(* IEC 61131-3 sources: ml2plc/benchmarks/st (part 15) *)

(* ---- MLP6.st ---- *)
FUNCTION_BLOCK MLP6_FB

    (* Model Inputs/Outputs *)
VAR_INPUT
    input_data : REAL;
END_VAR

VAR_OUTPUT
    output_data : ARRAY[0..2] OF REAL;
END_VAR

VAR CONSTANT
    weights_0 : ARRAY[0..31] OF REAL := [0.90454644, -0.400867403, 0.869943202, -0.168369889, -0.412142217, -0.709689677, 0.941532314, -0.0095654726, 0.967146814, -0.747319877, -0.0222444534, -0.66351074, -0.611298144, 1.09773886, -0.340438962, 1.20525312, 0.769771993, -0.182968155, -0.102920204, -0.384943873, -0.278610766, -0.314933598, 1.11625111, -0.168380052, -0.255054265, -0.366751343, -0.33793211, -0.02283746, 0.767741799, 0.474790365, 0.933169901, 0.962373257];
    bias_0 : ARRAY[0..31] OF REAL := [-0.170696706, 0, -0.161620259, 0, 0, 0.396536261, -0.158844277, 0, -0.152492061, 0.487909496, 0, 0.379839331, 0.448248148, -0.155945137, 0, -0.194220677, 0.0190808177, 0, 0, 0, 0, 0, 0.121851504, 0, 0, 0, 0.51204443, 0, -0.155369952, 0.399590701, -0.175982088, -0.155457303];

    weights_1 : ARRAY[0..767] OF REAL := [0.295231134, -0.129006118, 0.19198513, 1.21736336, -0.217146203, 0.906156719, -1.09466374, -0.706765652, 1.08418429, 0.564806283, 1.13035882, 0.892600179, -0.752894461, 1.10702014, 0.513110518, 0.785720646, -1.29299068, 0.0211936235, -1.44453084, -1.23774385, 1.08793128, -0.0487730801, -0.12848036, -1.00077665, 0.325005591, 0.290268898, 0.279054999, 0.285099328, -0.213655964, -0.16316177, 0.281590104, 0.239627063, 0.262345135, 0.0261963308, 0.0233350694, 0.294732571, 0.0434944928, 0.122584373, -0.150452822, -0.016712755, -0.261746407, -0.267375886, 0.240840673, -0.255916059, -0.249444306, 0.163675129, 0.0948724747, 0.162443012, 0.208322883, 0.238537252, -0.294643342, 1.23445666, -0.0170371439, 0.994598091, -0.975817561, -0.642093956, 1.19595969, 0.453583807, 1.12319052, 0.746419311, -0.853555024, 1.04991555, 0.597184777, 0.958240926, -1.17020535, 0.31369257, -1.47341204, -1.295645, 0.946281433, 0.27644223, -0.00174131989, -1.33688474, -0.176306188, -0.0927960575, 0.149620146, 0.286391616, -0.141670659, 0.0531999469, 0.153332919, 0.20505631, -0.167928115, 0.291448116, 0.150106311, -0.0987332314, 0.268482685, -0.307833642, 0.221213877, -0.321412444, 0.189507961, 0.191550195, 0.0819987059, -0.0778846443, 0.296701074, 0.225336492, 0.214712262, -0.0827709287, 0.285367191, -0.140551165, 0.00931853056, -0.138217196, 0.206591249, -0.0735297203, 0.221336126, 0.158516407, -0.0778366476, -0.271311015, 0.0633286238, -0.072303772, 0.108249843, -0.0929207653, -0.181190684, 0.0980706811, -0.0374506116, -0.320174545, 0.0739811957, -0.282686174, 0.186342359, 0.281644583, -0.259203553, 0.100598246, -0.0651429817, -0.206569076, -0.193545833, -0.482666612, -0.0821752772, -0.961810708, 1.172135, 0.69371134, -0.817266881, -0.412939996, -0.509167433, -0.866225541, 1.31189537, -0.633265257, -0.989419341, -0.846661031, 0.659452438, -0.225636706, 0.801334143, 0.350917637, -0.919107139, 0.225119472, -0.138609588, 0.721869826, -0.321482867, 0.123193502, 0.0898693502, 1.08808005, 0.295813471, 0.659393251, -0.476271152, -0.18717283, 1.23643327, 0.780925453, 0.986792803, 0.816414535, -0.891632259, 0.673117697, 0.646242201, 0.879625261, -0.865934372, -0.12343955, -1.18406153, -1.38234627, 0.901530623, 0.285107851, -0.256406724, -1.06379592, 0.107042551, 0.277778804, 0.193757594, 0.0590963066, -0.12765266, -0.133937359, -0.231395423, -0.289933264, 0.145242512, 0.23902446, 0.194817305, 0.0290448368, -0.0362384021, -0.17609328, 0.236915767, -0.0920998454, 0.252641916, 0.12115562, 0.000273287296, -0.269050717, -0.237204999, -0.219775066, 0.226729214, -0.231590211, -0.0661152154, -0.215537995, -0.235369325, 1.18310201, 0.173817322, 0.560130358, -0.859532833, -0.244359657, 1.11220109, 0.730377376, 0.526197612, 0.643959224, -0.431146711, 1.06084871, 0.894755185, 0.731103778, -0.696267724, 0.0121684372, -1.08033919, -1.12541819, 0.495167494, -0.101574555, 0.00402355194, -0.757044673, 0.136979058, 0.15508759, -0.02835216, -0.44361186, -0.275727361, -0.567569137, 0.871675193, 1.20000923, -0.853888154, -0.758741319, -0.443973094, -0.564651251, 1.32495701, -0.424292624, -0.405168772, -0.882857502, 0.919342339, -0.210148335, 0.787934899, 0.394117832, -0.723487794, -0.121570155, 0.274054289, 0.232991621, 0.184159577, -0.11905022, -0.173855618, 0.275910616, -0.213984191, 0.214573622, 0.247941315, -0.251989603, 0.207406044, 0.299859524, -0.0322960019, -0.235998034, -0.128714725, 0.137502581, -0.311281651, -0.0586145818, -0.236795753, 0.0351615846, -0.110103473, 0.0936356783, -0.203782856, 0.160411, -0.136357099, 0.217081785, -0.19382897, -0.0983214974, -0.172582373, -0.58115685, -0.227134705, -0.793690443, 0.987000167, 1.1088897, -0.533255935, -0.744200766, -0.41089806, -0.827442169, 0.908342123, -0.405829221, -0.716313243, -1.04521453, 0.604358673, -0.301062584, 0.378562003, 0.844146967, -0.835850179, 0.107833266, -0.223568857, 0.397432297, 0.188605264, -0.0674909353, 0.0566187575, 0.0197456405, 0.261059344, -0.524976611, 1.08699298, 1.06586397, -0.199344724, -0.802884936, -0.708495975, -0.716707826, 1.0185467, -0.364413172, -0.784771442, -0.431129128, 0.772798419, -0.185489476, 0.844132841, 0.761012673, -0.800541401, -0.0832273066, -0.2817581, 0.74396807, -0.264797121, -0.0910985023, -0.138044387, 0.990080476, 0.0802568346, 0.758434594, -0.552077353, -0.327732533, 0.887677908, 0.571260631, 0.937031686, 0.607444167, -0.378594458, 1.02893746, 0.491255462, 0.416121751, -1.0151366, -0.211483151, -0.746881902, -1.0333792, 0.443029851, -0.0171875358, -0.0381689072, -1.09573913, -0.043354094, 0.283042789, 0.206892252, 0.00916621089, -0.249695212, -0.295910805, 0.20259881, 0.162647396, 0.043733269, 0.20653832, -0.308564663, -0.280918926, 0.272660732, -0.172042117, 0.170747489, 0.23414731, 0.0630742013, 0.123369873, -0.207023829, 0.261101246, 0.213620901, 0.277589023, -0.0439403951, -0.205727562, 0.163603202, -0.113319919, -0.207964301, 0.628932774, -0.114935495, 0.705150783, -0.654717207, -0.237874627, 0.747101903, 0.727941096, 0.503591537, 0.72308296, -0.44854787, 0.965443373, 0.691107392, 0.5111745, -1.08201611, 0.21339798, -0.882919967, -1.20124686, 0.595513225, -0.252263993, 0.132210314, -1.06991637, -0.370881855, -0.0681702793, 0.169512168, 0.941228926, 0.070693031, 0.151429042, 0.256398469, 0.241526261, 0.751011312, 0.290890872, 0.30156377, 0.283818036, -0.0107974913, 0.482792228, 0.337298661, 0.281841606, -0.397284865, -0.208623588, -0.496294975, -0.470995426, 0.283237845, 0.0521007478, 0.144089073, -0.0686480999, -0.320380658, -0.277808845, 0.148536921, -0.0695285797, -0.277294815, -0.124862239, -0.0500250161, -0.222713381, -0.191136509, 0.246649325, 0.0220653415, 0.16214779, -0.061910063, 0.101160318, 0.157166272, -0.311789989, 0.000512182713, 0.0986146927, -0.171011031, 0.202872753, -0.215096593, -0.0623323619, -0.0904355496, 0.174473226, -0.301766038, 0.0454842746, -0.142736778, -0.020793587, -0.145345911, -0.178476349, 0.141361535, 0.0972788632, 0.110777199, 0.0764600039, 0.294599175, -2.27093697e-05, 0.173557222, 0.134258181, -0.311912924, -0.234820932, -0.187618434, -0.262826115, 0.192258656, 0.0524175763, 0.151788741, -0.03005898, 0.281539679, -0.157674417, -0.0799265057, -0.288467199, 0.0854136944, 0.153585076, 0.0907833874, -0.104148105, -0.0822955072, 0.210213959, 0.0297137201, -0.309015512, 0.0589160323, 0.156244159, -0.139795348, 0.276519597, 0.325013876, 0.0363880694, 0.127945542, 0.0618295372, -0.145081908, 0.192194581, 0.277251661, -0.144023046, -0.152517006, 0.231688559, -0.205610037, 0.22849232, 0.238232791, -0.29971382, 0.0167252421, -0.0997401178, -0.324124038, -0.127922207, 0.285681605, -0.10798724, -0.189939201, 0.294958234, -0.211431101, 0.211328328, -0.284518421, -0.18888253, -0.0722288787, -0.0350409448, -0.321308106, -0.0472274125, -0.0861286372, -0.316458166, -0.215742141, 0.0792055428, -0.0646136403, -0.274710715, -0.0250250399, -0.305008411, 0.229083359, 0.24799335, 0.0113067031, -0.249429077, -0.111249506, 0.237919688, -0.151925221, -0.318326861, -0.0953566432, 0.229551256, -0.163930863, 0.100224525, -0.167222232, -0.238116205, -0.202555746, -0.045360744, 0.0127826929, 0.280991137, -0.210080445, 0.0943366587, -0.0495974384, -0.0197191834, -0.149649471, 0.366648972, -0.281668693, 0.284846961, 0.403985202, 0.484802961, 0.784509182, 0.469572723, 0.473852932, 0.125889629, 0.312252492, 0.352212965, 0.477095902, -0.00642840099, -0.295710534, -0.206710175, -0.640399277, -0.231049523, 0.239183992, -0.311245203, -0.299947232, -0.0802108124, -0.0983978957, -0.173755497, -0.230084643, 0.316312313, -0.177855998, -0.298542112, 0.292203665, 0.00650158525, -0.297387481, -0.154374689, 0.162093848, 0.134812981, 0.246338308, 0.300070405, -0.310504198, -0.217782527, 0.0207454264, 0.0871799886, -0.264095902, 0.180105686, 0.285792828, 0.316828549, -0.150229871, 0.208020031, 0.136193275, -0.173812315, 0.0681842566, -0.221390352, 0.153097779, -0.194303483, 0.288291216, 0.12797904, 0.306318879, 0.212034047, -0.0300059021, 0.0768045485, -0.212660864, 0.171384782, 0.0894418657, -0.127920032, -0.21113494, -0.19953534, -0.211162567, 0.187122345, -0.174947098, -0.199379727, 0.0794975162, 0.270518363, 0.0516895354, 0.117571741, -0.0213138759, 0.146065593, -0.151934817, 0.324477196, 0.315924108, 0.0616651773, -0.300438493, 0.0912067592, -0.297835529, 0.13777557, 0.00982579589, -0.0171657801, -0.177937701, -0.210091144, 0.0937231779, -0.00284725428, -0.0512967706, -0.081265673, -0.277936608, 0.320349038, 0.0345208645, -0.0836495906, 0.218804076, -0.189922586, 0.00870514568, -0.0475570038, -0.215569362, -0.448498726, 0.7030285, 0.686182499, -0.145566911, -0.249483347, 0.0584986731, -0.39541024, 1.02209508, 0.23206374, -0.283743173, 0.0408624671, 0.087765269, 0.226524353, 0.406258434, 0.542207479, 0.000192098902, -0.154791355, -0.0193217993, 0.598222733, -0.155410215, -0.0176387131, -0.169864312, -0.207125589, -0.189757839, 0.0158335268, -0.170205817, 0.108427167, 0.163378179, 0.253302336, -0.147233725, -0.238223046, 0.0536537468, 0.00758227706, -0.275630891, 0.106042475, -0.240080804, -0.077775389, 0.144946277, -0.186762944, -0.104210451, 0.228787661, -0.0615751147, 0.211148441, -0.2518996, -0.019515574, 0.248782992, 1.05728996, -0.230006129, 0.742800951, -1.2359885, -0.62584269, 1.51240218, 0.719003975, 1.5774833, 0.910296917, -0.750651956, 1.05900729, 0.610199094, 1.06828773, -1.46972156, -0.31832701, -1.53218114, -1.44456565, 0.98592943, -0.268657327, -0.267539084, -1.16338086, -0.184921622, -0.0245098174, 0.181098208, 0.520282805, -0.0843829811, 0.0626276657, 0.461200267, 0.611355305, 0.621550381, -0.157471061, 0.200103998, -0.0395837352, 0.149573594, 0.173357353, -0.119783588, 0.0554200225, 0.0896117091, -0.160246953, 0.283200741, 0.299669445, -0.0905595943, -0.166233853, -0.0798888057, -0.229181871, 0.210135713, 0.0194011629, -0.0352008343, 0.728743076, 0.019356098, 0.761186361, -0.572355151, -0.597376704, 1.06806505, 0.662380099, 1.18272328, 0.938285351, -0.638570726, 0.836572111, 0.849231899, 0.980818689, -1.24159503, -0.29251948, -1.32303631, -1.02425313, 0.812224746, -0.230198115, 0.0245965719, -1.12541747, -0.0841034278, 0.118305951, 0.278894305, 1.19096649, 0.193239287, 0.558676004, -0.484399647, -0.12447723, 0.870661914, 0.808956504, 0.990534484, 0.965567052, -0.720074534, 0.667833567, 0.449974805, 0.92786181, -0.824072123, -0.092888996, -0.785955429, -0.710629821, 0.643768787, -0.179926112, -0.308975548, -0.589572847];
    bias_1 : ARRAY[0..23] OF REAL := [-0.041254133, 0, -0.00746029103, 0.0988344401, -0.0175108574, -0.163416371, 0.524258494, 0.51676178, 0.0377424657, -0.176874027, -0.0529647321, -0.118044838, 0.559266388, 0.0913945511, -0.158073679, -0.212183177, 0.239383668, 0, 0.26087296, 0.194069535, -0.150364339, 0, 0, 0.199199706];

    weights_2 : ARRAY[0..71] OF REAL := [-0.366981655, 0.407668054, -0.456144542, 0.0246128738, -0.193879545, 0.029107064, -0.161294922, 0.00702124368, -0.21840851, -1.41365981, 0.987270176, 0.742007971, -0.332335711, -0.0271744523, -0.441027492, -0.325576633, -1.88435066, 1.45009863, 0.876257122, 0.534476995, -1.14616477, 0.301283509, 0.361193687, -1.12447178, -1.20225334, 0.664745331, 0.887686074, -0.519799232, -1.71867156, 1.34296358, -1.97883332, 0.160939649, 0.910859942, -0.258056462, -1.82137454, 1.56507766, 0.472795397, 0.200812578, -1.2360208, -1.54919517, 0.81725806, 0.986340046, -0.0206529945, -1.71989512, 1.85158134, -0.0727280229, -1.53903365, 1.77559733, 1.76747835, -1.66802728, -0.428545892, -0.143300533, -0.339210212, 0.148096055, 1.281407, -2.03390622, -0.831091821, 1.72422087, -1.627334, -0.576684475, -0.803670168, -2.15200853, 1.69465089, 0.262259394, 0.242327183, 0.299449652, -0.337940395, -0.434468031, 0.11190328, 1.69577134, -2.20703983, -0.524324358];
    bias_2 : ARRAY[0..2] OF REAL := [0.173563749, 0.231935471, -0.377385825];

END_VAR

VAR
    (* Merged variables from all regions *)
    buffer_0 : ARRAY[0..23] OF REAL;
    buffer_1 : ARRAY[0..31] OF REAL;

    (* Temporary computation variables *)
    i : DINT;
    j : DINT;
    t : DINT;
    sum : REAL;
    (* Computation helpers *)
    max_val : REAL;
    exp_val : REAL;
    exp_sum : REAL;
    (* Spatial loop variables *)
    oc : DINT;
    oh : DINT;
    ow : DINT;
    ic : DINT;
    kh : DINT;
    kw : DINT;
    ih : DINT;
    iw : DINT;
END_VAR

(* Forward pass execution *)

(* Region: r0 [ACYCLIC] *)
(* Acyclic Region r0 *)
(* Layer 0: Fused Linear + RELU *)
FOR j := 0 TO 31 DO
    sum := 0.0;
    FOR i := 0 TO 0 DO
        sum := sum + input_data * weights_0[i * 32 + j];
    END_FOR;
buffer_1[j] := MAX(sum + bias_0[j], 0.0);
END_FOR;

(* Layer 1: Fused Linear + RELU *)
FOR j := 0 TO 23 DO
    sum := 0.0;
    FOR i := 0 TO 31 DO
        sum := sum + buffer_1[i] * weights_1[i * 24 + j];
    END_FOR;
buffer_0[j] := MAX(sum + bias_1[j], 0.0);
END_FOR;

(* Layer 2: Fused Linear + SOFTMAX *)
FOR j := 0 TO 2 DO
    sum := 0.0;
    FOR i := 0 TO 23 DO
        sum := sum + buffer_0[i] * weights_2[i * 3 + j];
    END_FOR;
output_data[j] := sum + bias_2[j];
END_FOR;

(* Softmax: find max *)
max_val := output_data[0];
FOR i := 1 TO 2 DO
    IF output_data[i] > max_val THEN
        max_val := output_data[i];
    END_IF;
END_FOR;

(* Softmax: compute exponentials and sum *)
exp_sum := 0.0;
FOR i := 0 TO 2 DO
    output_data[i] := EXP(output_data[i] - max_val);
    exp_sum := exp_sum + output_data[i];
END_FOR;

(* Softmax: normalize *)
FOR i := 0 TO 2 DO
    output_data[i] := output_data[i] / exp_sum;
END_FOR;

END_FUNCTION_BLOCK

(* ---- MLP6_straton.st ---- *)
FUNCTION_BLOCK MLP6_FB

    (* Model Inputs/Outputs *)
VAR_INPUT
    input_data : REAL;
END_VAR

VAR_OUTPUT
    output_data : ARRAY[0..2] OF REAL;
END_VAR

VAR
    CONSTANT weights_0 : ARRAY[0..31] OF REAL := [0.90454644, -0.400867403, 0.869943202, -0.168369889, -0.412142217, -0.709689677, 0.941532314, -0.0095654726, 0.967146814, -0.747319877, -0.0222444534, -0.66351074, -0.611298144, 1.09773886, -0.340438962, 1.20525312, 0.769771993, -0.182968155, -0.102920204, -0.384943873, -0.278610766, -0.314933598, 1.11625111, -0.168380052, -0.255054265, -0.366751343, -0.33793211, -0.02283746, 0.767741799, 0.474790365, 0.933169901, 0.962373257];
    CONSTANT bias_0 : ARRAY[0..31] OF REAL := [-0.170696706, 0, -0.161620259, 0, 0, 0.396536261, -0.158844277, 0, -0.152492061, 0.487909496, 0, 0.379839331, 0.448248148, -0.155945137, 0, -0.194220677, 0.0190808177, 0, 0, 0, 0, 0, 0.121851504, 0, 0, 0, 0.51204443, 0, -0.155369952, 0.399590701, -0.175982088, -0.155457303];
    CONSTANT weights_1 : ARRAY[0..767] OF REAL := [0.295231134, -0.129006118, 0.19198513, 1.21736336, -0.217146203, 0.906156719, -1.09466374, -0.706765652, 1.08418429, 0.564806283, 1.13035882, 0.892600179, -0.752894461, 1.10702014, 0.513110518, 0.785720646, -1.29299068, 0.0211936235, -1.44453084, -1.23774385, 1.08793128, -0.0487730801, -0.12848036, -1.00077665, 0.325005591, 0.290268898, 0.279054999, 0.285099328, -0.213655964, -0.16316177, 0.281590104, 0.239627063, 0.262345135, 0.0261963308, 0.0233350694, 0.294732571, 0.0434944928, 0.122584373, -0.150452822, -0.016712755, -0.261746407, -0.267375886, 0.240840673, -0.255916059, -0.249444306, 0.163675129, 0.0948724747, 0.162443012, 0.208322883, 0.238537252, -0.294643342, 1.23445666, -0.0170371439, 0.994598091, -0.975817561, -0.642093956, 1.19595969, 0.453583807, 1.12319052, 0.746419311, -0.853555024, 1.04991555, 0.597184777, 0.958240926, -1.17020535, 0.31369257, -1.47341204, -1.295645, 0.946281433, 0.27644223, -0.00174131989, -1.33688474, -0.176306188, -0.0927960575, 0.149620146, 0.286391616, -0.141670659, 0.0531999469, 0.153332919, 0.20505631, -0.167928115, 0.291448116, 0.150106311, -0.0987332314, 0.268482685, -0.307833642, 0.221213877, -0.321412444, 0.189507961, 0.191550195, 0.0819987059, -0.0778846443, 0.296701074, 0.225336492, 0.214712262, -0.0827709287, 0.285367191, -0.140551165, 0.00931853056, -0.138217196, 0.206591249, -0.0735297203, 0.221336126, 0.158516407, -0.0778366476, -0.271311015, 0.0633286238, -0.072303772, 0.108249843, -0.0929207653, -0.181190684, 0.0980706811, -0.0374506116, -0.320174545, 0.0739811957, -0.282686174, 0.186342359, 0.281644583, -0.259203553, 0.100598246, -0.0651429817, -0.206569076, -0.193545833, -0.482666612, -0.0821752772, -0.961810708, 1.172135, 0.69371134, -0.817266881, -0.412939996, -0.509167433, -0.866225541, 1.31189537, -0.633265257, -0.989419341, -0.846661031, 0.659452438, -0.225636706, 0.801334143, 0.350917637, -0.919107139, 0.225119472, -0.138609588, 0.721869826, -0.321482867, 0.123193502, 0.0898693502, 1.08808005, 0.295813471, 0.659393251, -0.476271152, -0.18717283, 1.23643327, 0.780925453, 0.986792803, 0.816414535, -0.891632259, 0.673117697, 0.646242201, 0.879625261, -0.865934372, -0.12343955, -1.18406153, -1.38234627, 0.901530623, 0.285107851, -0.256406724, -1.06379592, 0.107042551, 0.277778804, 0.193757594, 0.0590963066, -0.12765266, -0.133937359, -0.231395423, -0.289933264, 0.145242512, 0.23902446, 0.194817305, 0.0290448368, -0.0362384021, -0.17609328, 0.236915767, -0.0920998454, 0.252641916, 0.12115562, 0.000273287296, -0.269050717, -0.237204999, -0.219775066, 0.226729214, -0.231590211, -0.0661152154, -0.215537995, -0.235369325, 1.18310201, 0.173817322, 0.560130358, -0.859532833, -0.244359657, 1.11220109, 0.730377376, 0.526197612, 0.643959224, -0.431146711, 1.06084871, 0.894755185, 0.731103778, -0.696267724, 0.0121684372, -1.08033919, -1.12541819, 0.495167494, -0.101574555, 0.00402355194, -0.757044673, 0.136979058, 0.15508759, -0.02835216, -0.44361186, -0.275727361, -0.567569137, 0.871675193, 1.20000923, -0.853888154, -0.758741319, -0.443973094, -0.564651251, 1.32495701, -0.424292624, -0.405168772, -0.882857502, 0.919342339, -0.210148335, 0.787934899, 0.394117832, -0.723487794, -0.121570155, 0.274054289, 0.232991621, 0.184159577, -0.11905022, -0.173855618, 0.275910616, -0.213984191, 0.214573622, 0.247941315, -0.251989603, 0.207406044, 0.299859524, -0.0322960019, -0.235998034, -0.128714725, 0.137502581, -0.311281651, -0.0586145818, -0.236795753, 0.0351615846, -0.110103473, 0.0936356783, -0.203782856, 0.160411, -0.136357099, 0.217081785, -0.19382897, -0.0983214974, -0.172582373, -0.58115685, -0.227134705, -0.793690443, 0.987000167, 1.1088897, -0.533255935, -0.744200766, -0.41089806, -0.827442169, 0.908342123, -0.405829221, -0.716313243, -1.04521453, 0.604358673, -0.301062584, 0.378562003, 0.844146967, -0.835850179, 0.107833266, -0.223568857, 0.397432297, 0.188605264, -0.0674909353, 0.0566187575, 0.0197456405, 0.261059344, -0.524976611, 1.08699298, 1.06586397, -0.199344724, -0.802884936, -0.708495975, -0.716707826, 1.0185467, -0.364413172, -0.784771442, -0.431129128, 0.772798419, -0.185489476, 0.844132841, 0.761012673, -0.800541401, -0.0832273066, -0.2817581, 0.74396807, -0.264797121, -0.0910985023, -0.138044387, 0.990080476, 0.0802568346, 0.758434594, -0.552077353, -0.327732533, 0.887677908, 0.571260631, 0.937031686, 0.607444167, -0.378594458, 1.02893746, 0.491255462, 0.416121751, -1.0151366, -0.211483151, -0.746881902, -1.0333792, 0.443029851, -0.0171875358, -0.0381689072, -1.09573913, -0.043354094, 0.283042789, 0.206892252, 0.00916621089, -0.249695212, -0.295910805, 0.20259881, 0.162647396, 0.043733269, 0.20653832, -0.308564663, -0.280918926, 0.272660732, -0.172042117, 0.170747489, 0.23414731, 0.0630742013, 0.123369873, -0.207023829, 0.261101246, 0.213620901, 0.277589023, -0.0439403951, -0.205727562, 0.163603202, -0.113319919, -0.207964301, 0.628932774, -0.114935495, 0.705150783, -0.654717207, -0.237874627, 0.747101903, 0.727941096, 0.503591537, 0.72308296, -0.44854787, 0.965443373, 0.691107392, 0.5111745, -1.08201611, 0.21339798, -0.882919967, -1.20124686, 0.595513225, -0.252263993, 0.132210314, -1.06991637, -0.370881855, -0.0681702793, 0.169512168, 0.941228926, 0.070693031, 0.151429042, 0.256398469, 0.241526261, 0.751011312, 0.290890872, 0.30156377, 0.283818036, -0.0107974913, 0.482792228, 0.337298661, 0.281841606, -0.397284865, -0.208623588, -0.496294975, -0.470995426, 0.283237845, 0.0521007478, 0.144089073, -0.0686480999, -0.320380658, -0.277808845, 0.148536921, -0.0695285797, -0.277294815, -0.124862239, -0.0500250161, -0.222713381, -0.191136509, 0.246649325, 0.0220653415, 0.16214779, -0.061910063, 0.101160318, 0.157166272, -0.311789989, 0.000512182713, 0.0986146927, -0.171011031, 0.202872753, -0.215096593, -0.0623323619, -0.0904355496, 0.174473226, -0.301766038, 0.0454842746, -0.142736778, -0.020793587, -0.145345911, -0.178476349, 0.141361535, 0.0972788632, 0.110777199, 0.0764600039, 0.294599175, -2.27093697e-05, 0.173557222, 0.134258181, -0.311912924, -0.234820932, -0.187618434, -0.262826115, 0.192258656, 0.0524175763, 0.151788741, -0.03005898, 0.281539679, -0.157674417, -0.0799265057, -0.288467199, 0.0854136944, 0.153585076, 0.0907833874, -0.104148105, -0.0822955072, 0.210213959, 0.0297137201, -0.309015512, 0.0589160323, 0.156244159, -0.139795348, 0.276519597, 0.325013876, 0.0363880694, 0.127945542, 0.0618295372, -0.145081908, 0.192194581, 0.277251661, -0.144023046, -0.152517006, 0.231688559, -0.205610037, 0.22849232, 0.238232791, -0.29971382, 0.0167252421, -0.0997401178, -0.324124038, -0.127922207, 0.285681605, -0.10798724, -0.189939201, 0.294958234, -0.211431101, 0.211328328, -0.284518421, -0.18888253, -0.0722288787, -0.0350409448, -0.321308106, -0.0472274125, -0.0861286372, -0.316458166, -0.215742141, 0.0792055428, -0.0646136403, -0.274710715, -0.0250250399, -0.305008411, 0.229083359, 0.24799335, 0.0113067031, -0.249429077, -0.111249506, 0.237919688, -0.151925221, -0.318326861, -0.0953566432, 0.229551256, -0.163930863, 0.100224525, -0.167222232, -0.238116205, -0.202555746, -0.045360744, 0.0127826929, 0.280991137, -0.210080445, 0.0943366587, -0.0495974384, -0.0197191834, -0.149649471, 0.366648972, -0.281668693, 0.284846961, 0.403985202, 0.484802961, 0.784509182, 0.469572723, 0.473852932, 0.125889629, 0.312252492, 0.352212965, 0.477095902, -0.00642840099, -0.295710534, -0.206710175, -0.640399277, -0.231049523, 0.239183992, -0.311245203, -0.299947232, -0.0802108124, -0.0983978957, -0.173755497, -0.230084643, 0.316312313, -0.177855998, -0.298542112, 0.292203665, 0.00650158525, -0.297387481, -0.154374689, 0.162093848, 0.134812981, 0.246338308, 0.300070405, -0.310504198, -0.217782527, 0.0207454264, 0.0871799886, -0.264095902, 0.180105686, 0.285792828, 0.316828549, -0.150229871, 0.208020031, 0.136193275, -0.173812315, 0.0681842566, -0.221390352, 0.153097779, -0.194303483, 0.288291216, 0.12797904, 0.306318879, 0.212034047, -0.0300059021, 0.0768045485, -0.212660864, 0.171384782, 0.0894418657, -0.127920032, -0.21113494, -0.19953534, -0.211162567, 0.187122345, -0.174947098, -0.199379727, 0.0794975162, 0.270518363, 0.0516895354, 0.117571741, -0.0213138759, 0.146065593, -0.151934817, 0.324477196, 0.315924108, 0.0616651773, -0.300438493, 0.0912067592, -0.297835529, 0.13777557, 0.00982579589, -0.0171657801, -0.177937701, -0.210091144, 0.0937231779, -0.00284725428, -0.0512967706, -0.081265673, -0.277936608, 0.320349038, 0.0345208645, -0.0836495906, 0.218804076, -0.189922586, 0.00870514568, -0.0475570038, -0.215569362, -0.448498726, 0.7030285, 0.686182499, -0.145566911, -0.249483347, 0.0584986731, -0.39541024, 1.02209508, 0.23206374, -0.283743173, 0.0408624671, 0.087765269, 0.226524353, 0.406258434, 0.542207479, 0.000192098902, -0.154791355, -0.0193217993, 0.598222733, -0.155410215, -0.0176387131, -0.169864312, -0.207125589, -0.189757839, 0.0158335268, -0.170205817, 0.108427167, 0.163378179, 0.253302336, -0.147233725, -0.238223046, 0.0536537468, 0.00758227706, -0.275630891, 0.106042475, -0.240080804, -0.077775389, 0.144946277, -0.186762944, -0.104210451, 0.228787661, -0.0615751147, 0.211148441, -0.2518996, -0.019515574, 0.248782992, 1.05728996, -0.230006129, 0.742800951, -1.2359885, -0.62584269, 1.51240218, 0.719003975, 1.5774833, 0.910296917, -0.750651956, 1.05900729, 0.610199094, 1.06828773, -1.46972156, -0.31832701, -1.53218114, -1.44456565, 0.98592943, -0.268657327, -0.267539084, -1.16338086, -0.184921622, -0.0245098174, 0.181098208, 0.520282805, -0.0843829811, 0.0626276657, 0.461200267, 0.611355305, 0.621550381, -0.157471061, 0.200103998, -0.0395837352, 0.149573594, 0.173357353, -0.119783588, 0.0554200225, 0.0896117091, -0.160246953, 0.283200741, 0.299669445, -0.0905595943, -0.166233853, -0.0798888057, -0.229181871, 0.210135713, 0.0194011629, -0.0352008343, 0.728743076, 0.019356098, 0.761186361, -0.572355151, -0.597376704, 1.06806505, 0.662380099, 1.18272328, 0.938285351, -0.638570726, 0.836572111, 0.849231899, 0.980818689, -1.24159503, -0.29251948, -1.32303631, -1.02425313, 0.812224746, -0.230198115, 0.0245965719, -1.12541747, -0.0841034278, 0.118305951, 0.278894305, 1.19096649, 0.193239287, 0.558676004, -0.484399647, -0.12447723, 0.870661914, 0.808956504, 0.990534484, 0.965567052, -0.720074534, 0.667833567, 0.449974805, 0.92786181, -0.824072123, -0.092888996, -0.785955429, -0.710629821, 0.643768787, -0.179926112, -0.308975548, -0.589572847];
    CONSTANT bias_1 : ARRAY[0..23] OF REAL := [-0.041254133, 0, -0.00746029103, 0.0988344401, -0.0175108574, -0.163416371, 0.524258494, 0.51676178, 0.0377424657, -0.176874027, -0.0529647321, -0.118044838, 0.559266388, 0.0913945511, -0.158073679, -0.212183177, 0.239383668, 0, 0.26087296, 0.194069535, -0.150364339, 0, 0, 0.199199706];
    CONSTANT weights_2 : ARRAY[0..71] OF REAL := [-0.366981655, 0.407668054, -0.456144542, 0.0246128738, -0.193879545, 0.029107064, -0.161294922, 0.00702124368, -0.21840851, -1.41365981, 0.987270176, 0.742007971, -0.332335711, -0.0271744523, -0.441027492, -0.325576633, -1.88435066, 1.45009863, 0.876257122, 0.534476995, -1.14616477, 0.301283509, 0.361193687, -1.12447178, -1.20225334, 0.664745331, 0.887686074, -0.519799232, -1.71867156, 1.34296358, -1.97883332, 0.160939649, 0.910859942, -0.258056462, -1.82137454, 1.56507766, 0.472795397, 0.200812578, -1.2360208, -1.54919517, 0.81725806, 0.986340046, -0.0206529945, -1.71989512, 1.85158134, -0.0727280229, -1.53903365, 1.77559733, 1.76747835, -1.66802728, -0.428545892, -0.143300533, -0.339210212, 0.148096055, 1.281407, -2.03390622, -0.831091821, 1.72422087, -1.627334, -0.576684475, -0.803670168, -2.15200853, 1.69465089, 0.262259394, 0.242327183, 0.299449652, -0.337940395, -0.434468031, 0.11190328, 1.69577134, -2.20703983, -0.524324358];
    CONSTANT bias_2 : ARRAY[0..2] OF REAL := [0.173563749, 0.231935471, -0.377385825];
END_VAR

VAR
    (* Merged variables from all regions *)
    buffer_0 : ARRAY[0..23] OF REAL;
    buffer_1 : ARRAY[0..31] OF REAL;

    (* Temporary computation variables *)
    i : DINT;
    j : DINT;
    t : DINT;
    sum : REAL;
    (* Computation helpers *)
    max_val : REAL;
    exp_val : REAL;
    exp_sum : REAL;
    (* Spatial loop variables *)
    oc : DINT;
    oh : DINT;
    ow : DINT;
    ic : DINT;
    kh : DINT;
    kw : DINT;
    ih : DINT;
    iw : DINT;
END_VAR

(* Forward pass execution *)

(* Region: r0 [ACYCLIC] *)
(* Acyclic Region r0 *)
(* Layer 0: Fused Linear + RELU *)
FOR j := 0 TO 31 DO
    sum := 0.0;
    FOR i := 0 TO 0 DO
        sum := sum + input_data * weights_0[i * 32 + j];
    END_FOR;
buffer_1[j] := MAX(sum + bias_0[j], 0.0);
END_FOR;

(* Layer 1: Fused Linear + RELU *)
FOR j := 0 TO 23 DO
    sum := 0.0;
    FOR i := 0 TO 31 DO
        sum := sum + buffer_1[i] * weights_1[i * 24 + j];
    END_FOR;
buffer_0[j] := MAX(sum + bias_1[j], 0.0);
END_FOR;

(* Layer 2: Fused Linear + SOFTMAX *)
FOR j := 0 TO 2 DO
    sum := 0.0;
    FOR i := 0 TO 23 DO
        sum := sum + buffer_0[i] * weights_2[i * 3 + j];
    END_FOR;
output_data[j] := sum + bias_2[j];
END_FOR;

(* Softmax: find max *)
max_val := output_data[0];
FOR i := 1 TO 2 DO
    IF output_data[i] > max_val THEN
        max_val := output_data[i];
    END_IF;
END_FOR;

(* Softmax: compute exponentials and sum *)
exp_sum := 0.0;
FOR i := 0 TO 2 DO
    output_data[i] := EXP(output_data[i] - max_val);
    exp_sum := exp_sum + output_data[i];
END_FOR;

(* Softmax: normalize *)
FOR i := 0 TO 2 DO
    output_data[i] := output_data[i] / exp_sum;
END_FOR;

END_FUNCTION_BLOCK

(* ---- MLP7.st ---- *)
FUNCTION_BLOCK MLP7_FB

    (* Model Inputs/Outputs *)
VAR_INPUT
    input_data : REAL;
END_VAR

VAR_OUTPUT
    output_data : ARRAY[0..2] OF REAL;
END_VAR

VAR CONSTANT
    weights_0 : ARRAY[0..23] OF REAL := [-0.0746802986, 0.607636034, 0.455998242, 0.258762628, -0.13258031, 0.252115637, -0.10976994, 0.548266053, -0.441276819, -0.438432246, 0.647188544, 0.493570745, -0.43271625, -0.082831949, 0.649822593, 0.439375341, -0.287549376, -0.311959922, 0.274157524, 0.315673918, 0.643515408, -0.171732515, 0.496268243, -0.371054083];
    bias_0 : ARRAY[0..23] OF REAL := [0, -0.12941812, -0.105221123, -0.0604603514, 0, 0.207637087, 0, 0.0315683261, 0, 0, -0.117396198, -0.0605233088, 0, 0, 0.0510026328, -0.0530445352, 0, 0, -0.0639983788, 0.203389689, -0.111548714, 0, -0.0640599579, 0];

    weights_1 : ARRAY[0..575] OF REAL := [-0.268907338, 0.00217190385, 0.137464732, -0.0683488548, -0.0738091469, 0.0699335039, -0.0417425632, 0.19087711, 0.0489356816, 0.344365627, 0.157603174, 0.211316198, -0.259004354, -0.257717103, 0.277782112, 0.273165613, 0.265473157, -0.205595359, 0.217125148, 0.343775719, 0.000431239605, -0.204861492, -0.16889219, -0.295836747, -0.612856627, -0.141135335, 0.4472965, -0.0880493671, -0.0630476475, -0.510043383, 0.529629707, 0.314925313, -0.324320614, -0.509671628, 0.322658747, 0.241676986, 0.696524978, 0.524104714, -0.213002667, 0.243135035, -0.297149271, -0.177744299, -0.219710499, 0.546750069, 0.511470258, 0.148470536, 0.587771058, 0.699641109, -0.699686229, -0.0136144357, 0.265989453, 0.187910274, 0.342317551, -0.476634353, 0.119458191, -0.123250976, 0.135319307, -0.525157869, -0.262663037, 0.386619776, 0.15526025, 0.15252319, 0.0138672292, 0.709074318, -0.214552373, 0.198164448, -0.329590023, 0.262734801, 0.253178746, 0.00747139985, 0.705926538, 0.132839769, -0.604175448, 0.0361758061, 0.386252105, 0.259136945, 0.121620715, -0.502793372, 0.120056905, 0.172273502, 0.197177142, -0.220736131, 0.312253743, 0.319560826, 0.478767067, 0.399403363, 0.299865872, 0.712916255, 0.00703683496, -0.358783484, -0.118123114, 0.141307041, 0.27085793, -0.305572391, 0.74335593, 0.179063112, -0.300123811, 0.294067651, 0.277188748, -0.273958385, -0.176085144, -0.0395295322, 0.172060519, -0.157897264, -0.331464142, -0.019657284, 0.114273429, 0.14408347, 0.0497518182, -0.119545832, -0.169999823, -0.30714044, -0.0324544311, 0.29038915, 0.094248265, 0.210150927, 0.158477634, -0.136283606, -0.0214261115, 0.0398223698, 0.216942891, -0.0235428363, 0.118681543, 0.083537966, -0.249544412, 0.332191288, 0.358593881, -0.315374881, 0.236496851, 0.186359823, -0.021189332, 0.485366553, -0.218409613, -0.00703188404, -0.112409517, -0.153913006, 0.210461989, 0.118319869, 0.173140079, 0.35994482, 0.224077418, 0.377764165, 0.135184735, 0.0969982445, 0.0219076872, -0.319111407, 0.0442451835, 0.314922959, 0.342028826, 0.154806107, -0.251459479, 0.231669575, 0.166534096, -0.14645718, -0.199890018, 0.29779157, 0.181536824, 0.22370407, 0.147348255, -0.241052836, 0.276352018, 0.0678429306, -0.271346122, -0.32665199, -0.179163054, 0.057913214, -0.216329142, -0.161545247, 0.236314058, 0.198999107, 0.204323336, 0.109188184, 0.185613602, -0.00481222663, -0.108478963, -0.184006527, -0.16169177, -0.126572222, -0.182018921, 0.401931792, 0.0411342047, 0.274655849, -0.312093377, 0.0779248402, -0.244552612, -0.0933865234, -0.143112406, 0.316888869, -0.0897234753, 0.444688708, 0.0414355583, 0.468671679, 0.224688619, -0.106085896, 0.12706238, 0.0274204016, -0.269548059, 0.0074904263, -0.25059554, -0.250605166, 0.317630261, 0.123651862, -0.246514887, 0.168738812, 0.28361252, 0.119744748, 0.141637355, 0.193590432, 0.245099097, -0.271869928, 0.305476636, 0.214189082, 0.0639041364, -0.251134604, -0.280500591, -0.182719231, 0.0889582634, 0.106302857, 0.308100551, -0.123537555, 0.155842453, 0.0435905457, 0.282452852, 0.0464273691, -0.329868048, 0.189582318, 0.0826188624, 0.268325478, -0.282127619, 0.325057715, 0.0578409731, -0.106060609, 0.122288734, 0.281878263, 0.0715391338, 0.0967436135, 0.312681288, 0.346843749, 0.286530644, 0.323031157, -0.62107712, 0.31202659, 0.439596415, -0.344784915, -0.217742249, -0.058255773, 0.255871952, 0.122528382, 0.234015152, 0.190027699, 0.0680105984, 0.477807403, 0.580108285, 0.111387841, 0.32501927, 0.465298355, 0.0707894638, 0.211896211, 0.313886732, 0.0590125956, 0.536113501, -0.110482946, 0.383503079, 0.321528226, -0.391103178, -0.0757583752, 0.477379769, -0.0182638038, -0.226764709, -0.114267945, 0.544339299, 0.341566026, 0.204276666, -0.276710838, -0.0310451984, 0.337987483, 0.101955645, 0.466226697, 0.00610649586, 0.0666570589, 0.251989096, -0.0348885134, -0.029322058, 0.0374343842, 0.548539996, 0.448163837, -0.0839401558, 0.467522532, -0.0633949339, 0.207616359, 0.0878649652, 0.00687465072, 0.266888529, 0.191955179, -0.319217205, 0.33818987, 0.0626723766, -0.093282342, 0.290955514, -0.015552938, -0.147785395, -0.222969472, 0.000421226025, 0.087808311, -0.184572592, -0.030451268, 0.308537692, 0.324173838, -0.0962346494, -0.0917209089, 0.121005028, 0.0796872079, 0.212975711, -0.169214532, -0.0300399065, 0.26500538, 0.0404863358, 0.188591808, -0.195912629, 0.175725371, -0.119754195, -0.180573285, -0.260601789, 0.318698615, 0.0112495124, 0.332248241, -0.0760537386, -0.140548617, 0.0673505664, 0.277959973, -0.230266511, -0.304319382, -0.0186672509, -0.289335996, 0.174558014, -0.0480471551, 0.156338379, -0.338227391, 0.379409701, -0.329904109, -0.0335883498, -0.0243462808, 0.106674857, -0.207976103, -0.31758371, -0.205548838, -0.286922336, 0.453636765, 0.344143778, -0.139424697, 0.150888771, 0.368412137, -0.0207992848, 0.433938384, -0.227954015, 0.451291412, 0.0406967625, 0.444359481, 0.183337077, 0.00309645641, 0.182288632, 0.142382234, -0.138220325, -0.0159723535, -0.266371191, -0.157991484, 0.509245634, -0.3441737, -0.300116122, -0.289941072, -0.25277108, 0.275200456, 0.381681621, 0.368882239, 0.191403657, 0.299521059, 0.0331215486, 0.0199813955, 0.0838560462, -0.0338563249, 0.552538455, -0.0257612541, 0.162927568, 0.157294571, -0.0424414575, 0.0741851032, 0.00993341208, 0.14510569, -0.19807291, -0.216219321, -0.326386631, -0.0369665921, -0.350637496, 0.327333599, 0.187157542, -0.191772714, -0.272784531, 0.178999513, 0.170922011, 0.344064087, 0.273409277, -0.195383936, 0.0219087601, -0.320345551, -0.223053589, -0.167534485, -0.353014231, -0.0325659513, 0.133774012, 0.300787896, -0.154813468, -0.109787136, 0.0450620651, -0.120923176, -0.126991063, -0.150874168, 0.330428869, -0.0456075966, 0.0592706203, 0.153212577, -0.167818964, -0.31344831, -0.313499629, 0.0622265339, -0.132025421, -0.0950550437, -0.172515988, -0.309438348, -0.241304442, 0.0670445859, 0.340844244, -0.00674307346, -0.0571297407, 0.195944682, 0.291546017, -0.089925617, -0.17480801, -0.509736598, 0.418891937, 0.187606826, -0.153403401, -0.149088994, 0.208767861, -0.081951119, 0.658967853, 0.617743134, -0.0702296197, 0.572496474, 0.191262931, 0.193394378, -0.252258331, 0.573703945, 0.182828963, -0.104402117, 0.189143315, 0.72547698, 0.252746373, -0.127337083, 0.359964609, 0.252452195, 0.0182416737, 0.158887416, 0.348938584, -0.0390769318, 0.164680511, 0.340248942, -0.29226917, -0.0991819948, 0.165644377, -0.00725150527, -0.105002299, -0.112420052, -0.139867827, 0.569023848, -0.310940892, 0.0389346555, 0.177371755, 0.124769427, 0.120482311, -0.127293751, 0.0575004928, -0.217616215, 0.0183300879, 0.123401649, 0.098418802, -0.383335978, 0.410907269, -0.0536490418, -0.247322127, -0.27997908, 0.27313289, 0.325315207, 0.4671942, 0.590981603, -0.332647026, 0.412228435, -0.349655986, -0.245886207, -0.194440514, 0.346960187, 0.216047853, 0.107523225, 0.0693727285, 0.547360241, -0.303221017, -0.0726420283, -0.102691054, 0.24672243, 0.184002489, -0.106598735, -0.143918335, 0.0378342271, 0.105892092, -0.0521823466, -0.241860956, 0.0522222221, 0.290780276, 0.329312891, -0.0297322273, 0.299719065, -0.0803425908, -0.127563834, -0.258438736, 0.128532708, 0.0761955082, 0.202705115, -0.275218487, 0.284864634, -0.285524696, 0.23296684, 0.558344007, -0.370309085, 0.0632788539, -0.199879572, 0.378469765, 0.168243155, -0.204663306, -0.111090496, -0.0149026215, 0.482993186, 0.230562359, -0.0151113905, -0.081802994, 0.302559614, 0.28712967, 0.350448579, 0.287046105, 0.0832951739, 0.450847089, 0.149081931, 0.352454573, 0.548047662, -0.231863469, 0.299252719, -0.0325100422, -0.237312376, 0.0971217752, -0.00699299574, 0.248950452, -0.0907193124, -0.16760385, 0.145382762, 0.0910830498, -0.00387185812, -0.277013451, 0.126328528, -0.23418954, -0.0778735578, -0.27938059, -0.349283576, 0.0730948448, 0.255102366, 0.0797807872, 0.0635040104, 0.0545716584, 0.144961387];
    bias_1 : ARRAY[0..23] OF REAL := [0.176716387, -0.00299654785, 0.0593073107, -0.0575258322, 0, 0.129074454, -0.103701882, -0.0082479585, -0.0571199395, 0.0882943869, 0, 0.208057463, -0.135922343, -0.0881750807, 0, -0.0836111233, -0.00893536955, 0.244989246, 0, -0.100842871, 0.0560074486, 0.252564728, -0.143066466, -0.12537545];

    weights_2 : ARRAY[0..575] OF REAL := [-0.245642945, -0.246756554, -0.328891218, -0.563465476, -0.555797517, 0.0490016043, -0.233312637, -0.150199234, 0.353149563, -0.227947727, 0.0115364343, 0.158489317, 0.142654747, -0.431395471, 0.344945014, 0.324086517, 0.612027287, -0.219665155, -0.0898557678, 0.145038947, 0.593772233, -0.217062712, -0.195034459, -0.363241315, 0.119104199, 0.22720471, -0.0466149151, -0.0383172072, -0.331802279, 0.343306452, -0.171254784, 0.156157047, 0.276797444, 0.220166475, -0.158973664, 0.32375142, 0.0450913534, -0.326723188, -0.201807857, 0.308251947, 0.226838693, 0.0587440133, 0.245269522, 0.266734153, 0.1890876, 0.0765732601, -0.0288925171, 0.223519564, 0.280389965, 0.0145830512, 0.00144499971, 0.139997378, 0.113765299, -0.191146329, 0.307509392, 0.179293185, 0.374915421, 0.30121091, 0.495148122, 0.0815368593, 0.434390634, -0.14555715, 0.433478117, -0.190034807, -0.0800786242, -0.200110286, 0.509086668, 0.318211406, 0.302050829, 0.0287599247, 0.141590983, 0.31887728, -0.226454079, 0.348596007, -0.016703397, 0.173407003, -0.270399421, 0.0868661702, -0.156372473, -0.12866497, 0.372414291, 0.347522587, 0.182157025, 0.241545171, -0.323187351, -0.271822125, -0.0328329206, -0.257270426, 0.004878846, -0.164576188, 0.32456243, 0.324977875, -0.0877593905, 0.244203418, 0.17296055, -0.27077353, -0.148512006, 0.0627348125, -0.235144854, 0.224023789, 0.258846492, 0.190566212, -0.136538416, 0.244612128, -0.260796845, -0.264053375, 0.20704934, 0.112125605, 0.108366191, 0.0839831531, -0.248119086, 0.210814208, -0.126879886, -0.19144927, -0.0575715005, -0.315923661, 0.152904361, -0.107165188, 0.098418355, -0.281930566, -0.0221283156, -0.242865384, 0.147830218, -0.0177736022, -0.0663293079, -0.191042975, -0.139932171, -0.0271336436, 0.306826115, 0.108970776, -0.47794044, 0.289082974, 0.848751605, -0.043951571, 0.271782011, 0.565594852, 0.176920876, 0.293638378, -0.185994714, -0.183791861, 0.492481083, -0.160842761, -0.195042297, -0.15548411, 0.224055469, 0.200847, -0.0932983235, 0.251617342, 0.455671281, 0.261954457, -0.0860045254, -0.0112277567, 0.242849126, -0.0363826528, 0.0945869535, -0.158523649, 0.232608065, 0.18994756, 0.048118569, 0.226275221, -0.00935058389, -0.233899072, -0.0633342341, 0.261702985, 0.00170290633, 0.43676585, -0.244740173, 0.53414011, 0.204737216, -0.0611152947, -0.105342865, -0.0732150078, 0.120023869, 0.261113197, 0.138036996, 0.333630413, 0.250143796, -0.0457339585, 0.214532509, -0.307090104, -0.333172113, 0.0266219284, -0.334947944, 0.0495177507, -0.121425427, 0.226054937, 0.281170636, 0.107468642, 0.277073115, -0.225816518, -0.219915509, -0.15749234, 0.184502214, -0.273863554, 0.233854562, -0.0685526431, -0.291586995, 0.0733211935, -0.303754866, 0.266844183, 0.311533213, 0.295593113, 0.183031395, 0.138876736, -0.298650354, 0.187308699, 0.158070579, -0.038877558, -0.0276067965, -0.141152993, 0.110567927, -0.232558206, -0.186817855, 0.0793989003, -0.158586457, 0.22946766, -0.501852512, -0.299868256, 0.256566316, -0.582294166, -0.448347151, -0.210635707, 0.322008342, -0.258173883, 0.379928738, 0.275341272, 0.199535474, -0.322017342, 0.800383627, -0.195558012, 0.220077574, 0.16850391, 0.0875466466, -0.137633145, -0.405929536, 0.0637919232, 0.397787511, -0.118515283, -0.0634722114, -0.508549154, -0.318264753, -0.0369980335, 0.339129716, -0.185298115, 0.318987221, -0.257021844, 0.326296836, -0.125292212, 0.215666503, 0.00417363644, -0.105437919, 0.0311455131, -0.263626844, 0.0762697756, -0.0561151505, 0.2861332, -0.207532167, 0.3018938, 0.0366989374, 0.210771888, -0.133724362, 0.0648821294, 0.0861230493, -0.151588723, 0.165128812, -0.318110764, 0.0824543834, 0.410491556, -0.16636388, -0.265668929, -0.217291281, -0.280920208, 0.376858443, -0.303223848, 0.448855996, -0.170281783, 0.354806125, 0.0322148241, 0.419946581, -0.099502638, 0.0150394971, -0.224528477, 0.499678612, 0.0742175803, 0.185917586, 0.272458673, -0.24160108, -0.0894065127, 0.669480681, -0.0906793773, 0.0840942785, 0.293848902, 0.649855793, -0.118749589, -0.319913119, 0.00412905216, -0.229158893, 0.131725997, 0.490128577, 0.209284037, -0.309097946, 0.35574317, 0.25872305, -0.335510433, -0.425682485, -0.228162214, 0.511070549, 0.0847743154, -0.507714033, 0.37029779, -0.130451664, 0.461581945, 0.503590107, -0.0959527791, -0.10381075, 0.129085854, 0.118843004, -0.0449370444, 0.265093714, 0.138016343, -0.413666576, 0.185948581, 0.289212912, -0.0518284738, -0.188458264, 0.396242261, -0.00943513215, -0.649417937, -0.62592417, 0.00135046244, 0.452810377, 0.501355469, -0.709819973, 0.628315389, 0.343882769, 0.65114969, -0.0102708638, -0.16960068, 0.320089728, 0.325349718, -0.327407748, 0.243835896, -0.0235780478, 0.210580379, 0.239429086, -0.0277884305, 0.245251507, -0.0667792261, 0.0719113648, 0.226514786, -0.228350446, -0.214209169, 0.0621877611, 0.307303458, -0.116270259, -0.338030607, -0.0395987332, -0.278134644, -0.0744503736, 0.297008485, 0.393869758, 0.33913973, 0.12972188, 0.293395817, 0.713052988, 0.037013948, -0.172523066, 0.0210779905, -0.549971342, 0.0169248395, 0.0676543564, -0.078420192, -0.274449199, 0.307433218, 0.00872946065, -0.376850694, -0.411587656, 0.106564432, 0.32417807, 0.567158878, -0.647322595, 0.517194271, 0.351190478, 0.386148691, 0.324564457, -0.349219918, 0.0146075785, 0.341831416, 0.135289431, -0.112718031, -0.0742655993, -0.150912598, 0.157066315, 0.242844671, -0.358709872, -0.0578418374, 0.139578655, -0.303983897, -0.0327897929, -0.0647751093, 0.109798618, -0.236207291, 0.0410545506, 0.228533059, -0.179919437, 0.174975157, 0.00423380733, 0.31155178, -0.151971802, -0.119472831, -0.304712266, 0.266190737, 0.333312094, 0.0527635515, -0.339556247, -0.308178425, 0.0686535835, -0.0389595479, 0.467055798, -0.0529330671, 0.566560745, 0.0217954665, 0.0637522563, 0.394496739, 0.175899759, 0.0786572993, 0.533386767, 0.222399384, 0.458613098, 0.00105759059, -0.0628268719, -0.171422854, 0.252415031, 0.173769027, 0.183591932, 0.247483999, -0.144038543, 0.318444401, -0.0695573986, -0.234271988, -0.0879763961, 0.272262067, -0.310317963, -0.164369002, 0.0924783647, -0.139321119, -0.183811679, -0.263402045, 0.347119004, -0.141531646, 0.115062743, 0.0182715952, 0.221911341, 0.188233048, 0.107228249, 0.156428427, 0.249304071, 0.339434177, 0.232620925, -0.0617873147, 0.0977720171, -0.220434427, 0.105078757, -0.221959457, -0.170278221, -0.0669473931, 0.319006234, 0.118522257, 0.324670047, 0.485926092, -0.00689097121, 0.15161325, 0.21309416, -0.255844951, 0.167315274, 0.544760644, -0.292000622, 0.306418985, -0.307936668, 0.186714277, 0.0277817752, -0.329396993, -0.371986449, 0.42815277, 0.0916256607, -0.181429625, -0.33743602, -0.0793887377, -0.259026438, -0.0198467597, 0.422208548, -0.207560241, 0.232187256, 0.478278846, 0.335845023, 0.0116891321, 0.233216554, -0.34780556, 0.456520617, 0.0233263914, 0.187153757, 0.307537764, -0.00473511219, 0.149918661, -0.00606621895, 0.00571098924, -0.207502544, -0.183465093, 0.298180431, 0.045966208, 0.0130442083, -0.175817266, 0.410728335, 0.185252845, -0.105908722, -0.135901928, 0.595315337, 0.128219843, 0.53443414, 0.37661013, 0.135160387, 0.0851265192, 0.129262373, 0.0782697424, 0.110159196, 0.209644005, -0.0161204934, 0.242139533, 0.351693124, 0.111278623, -0.0508820266, 0.151348934, 0.249107957, 0.325930446, -0.113416329, -0.0454256237, -0.415055484, -0.360494643, 0.349898517, 0.238396317, 0.146553114, 0.142856315, -0.136616945, -0.479777694, -0.573965073, -0.229324624, 0.105782844, 0.423111051, -0.526070297, 0.434536278, 0.029494375, 0.565732479, 0.583604753, -0.277379364, 0.265477479, 0.166019455, 0.326392949, -0.0792272985, -0.311522603, 0.253521353, -0.380653828, -0.0587646104, -0.0119071128, -0.311399788, 0.331956893, 0.620487213, 0.00493989419, -0.590279043, -0.207389817, -0.0455776751, 0.283825159, 0.635202348, -0.238840938, 0.540888488, -0.0559566915, 0.207977518];
    bias_2 : ARRAY[0..23] OF REAL := [-0.104559369, 0, -0.0181077477, -0.137459263, -0.135881066, 0, 0, 0, 0.142547369, -0.0255238134, 0.0494711883, 0, 0.260531038, -0.139503524, 0.25024417, 0.189121932, 0.195312738, 0, 0.0421190374, -0.0893590972, 0.201172814, -0.0583064407, 0, -0.115013145];

    weights_3 : ARRAY[0..575] OF REAL := [-0.602241993, 0.55888021, -0.167094216, 0.0352712572, 0.198801786, -0.316523612, 0.665048659, -0.343073666, 0.181268543, 0.0253115129, 0.255773276, 0.412630647, 0.149497539, -0.3257626, 0.561596334, -0.427766412, 0.612147987, -0.112615697, -0.0723482892, 0.0113181919, 0.207391828, 0.412549496, -0.283578128, -0.278952479, 0.0597497225, -0.28283149, -0.0710432231, 0.145420283, -0.106071651, 0.09520787, 0.120398045, -0.342419535, -0.130383208, -0.00268754363, 0.0910975337, -0.135052741, 0.239594012, 0.125919849, 0.239025921, 0.225845069, 0.000677734613, -0.130891666, -0.0202915072, -0.17219685, -0.249355674, -0.348977596, -0.332513243, 0.18060413, -0.262752742, 0.0582385957, -0.219546899, -0.194849432, -0.170968443, -0.0450304598, -0.267174065, 0.0574418604, 0.303428322, -0.0240614004, -0.0952934325, -0.191922903, -0.146774873, 0.223994285, 0.057148084, 0.302169144, -0.32576865, -0.304440975, -0.108279869, -0.158450708, -0.0436111987, 0.0403712541, -0.309476197, -0.0396765359, -0.391235322, 0.00788531173, -0.254363298, -0.160379454, -0.0967926681, -0.250588834, 0.18227306, -0.199728549, 0.151370078, 0.554630756, -0.315505922, 0.572615266, 0.0212666988, -0.112852648, 0.0755843297, -0.307928711, 0.455886036, 0.168461785, 0.0398970768, -0.426429212, 0.0424583852, 0.478647113, -0.153755188, -0.421815217, -0.409806162, 0.510546744, -0.0551810861, -0.0795919597, -0.00575041352, 0.134758815, 0.507890344, -0.2852723, -0.331913263, 0.117690071, -0.0528320968, 0.553075373, -0.242619514, -0.294256479, 0.634651184, -0.143082932, -0.0406088158, -0.0395390503, -0.20047991, -0.561169028, -0.0722154081, 0.532352924, -0.0981325209, -0.398828059, -0.0395203531, -0.269496202, 0.0321588814, -0.215388343, 0.238568455, 0.33127448, -0.125521317, 0.242836207, 0.0522266924, -0.29994604, 0.152543455, 0.225400239, -0.171876103, 0.129318833, -0.235493153, -0.00765952468, 0.237490684, 0.260011584, 0.0333464146, -0.00917688012, -0.00841370225, 0.10748744, -0.00466170907, -0.278230488, 0.189867824, -0.281087369, -0.274116457, -0.140237644, -0.283562392, -0.303457975, -0.105420902, -0.08898893, 0.324018449, -0.0211086571, -0.0984889269, 0.134744555, -0.100908309, -0.259068429, -0.14006266, 0.132343978, 0.28123638, -0.167043716, -0.177914992, 0.20753023, 0.323781103, -0.267359883, -0.0927713513, -0.29192549, -0.0374050736, -0.0302143991, -0.272224218, 0.0217229128, 0.156398922, 0.319664091, 0.252935201, 0.161032051, 0.309321433, -0.317337781, -0.127192274, -0.205821097, 0.350479096, 0.221662313, -0.198564246, -0.19292897, 0.146428674, -0.311415642, 0.323936731, -0.207948253, 0.183813423, -0.15229629, 0.21302703, 0.00983792543, -0.0352235399, 0.0982181355, 0.329058379, 0.0777703822, -0.244565234, 0.0349554829, 0.135095939, -0.238787457, 0.105752438, 0.0180288199, 0.00903719664, 0.142666906, -0.176260218, 0.0678556859, -0.0808573142, 0.1865215, -0.280900449, -0.312621117, -0.234703735, 0.543368936, -0.0145166516, 0.241052374, 0.093909122, 0.371220917, -0.0340538584, 0.0553505681, 0.00168967247, 0.00688350201, 0.016012013, 0.134655029, 0.104506545, 0.351621717, -0.197626323, 0.305818617, 0.194396943, -0.244596228, 0.0998549759, -0.0224575996, -0.0106034633, 0.305570573, -0.321722865, 0.116607845, -0.2247715, 0.329801023, -0.11524196, -0.29490301, 0.207909733, -0.00686628604, 0.0063027516, -0.0837529153, 0.14334321, 0.212508291, 0.161416039, 0.0928216651, 0.430584371, 0.299479485, -0.0385227203, 0.257451743, -0.0911267102, -0.122735053, -0.252591699, -0.150701806, 0.34466657, 0.393089354, 0.210057423, -0.157372728, 0.163869187, 0.159027457, -0.238099173, 0.364011973, -0.354819804, -0.141737163, 0.332482427, 0.00705638528, -0.286498755, 0.255034357, -0.217193916, -0.163846552, 0.0951987803, -0.0458124578, -0.0418757498, -0.245432392, -0.0318156481, -0.228291094, -0.122520894, -0.278282046, -0.150279894, 0.179519027, 0.211612433, 0.214148492, 0.0416107476, 0.126119971, -0.0671995282, -0.10378173, 0.331519514, -0.0976586342, 0.240162462, 0.061647296, -0.0112053156, -0.225412548, -0.231608272, 0.174605906, 0.226156548, -0.0398120768, -0.318600833, 0.583029628, -0.297376931, -0.0821852535, -0.158475772, 0.289350927, 0.15018031, 0.208243743, 0.142259523, 0.169374242, 0.325451702, 0.375857145, 0.0847464502, 0.486003429, 0.219020039, 0.347213596, -0.498953462, 0.575930357, -0.286445409, 0.201231569, -0.26902625, 0.193424612, 0.665235519, -0.281682044, -0.273364455, 0.422559619, 0.226529211, 0.228482798, -0.16290246, -0.140528128, 0.273387074, -0.344221294, 0.542001069, 0.108456314, -0.292378485, -0.450960845, -0.11324732, 0.300137132, 0.233597487, -0.0970329121, 0.150379717, -0.0796741471, -0.0803582668, 0.319187373, 0.256698847, 0.203733876, -0.025490975, -0.197300538, 0.000113457441, 0.378923118, -0.214601964, 0.261108875, -0.0262481272, -0.19515121, -0.0206418242, 0.205336094, 0.0494867563, 0.0813631341, 0.0376687236, 0.152586415, 0.101950288, 0.454461485, -0.228070661, 0.415039688, 0.204862505, -0.157589823, -0.282065004, 0.204876691, -0.0521092713, -0.30861786, -0.523558199, -0.0130606955, -0.061824441, -0.00745187514, 0.148885161, -0.37855342, 0.113599747, -0.243788734, 0.0348514281, 0.443149805, -0.182924971, -0.294054627, -0.258397967, 0.40322265, -0.0105616748, 0.121344253, -0.202887818, 0.46591261, 0.488460571, -0.406302303, -0.0231820345, -0.208175167, -0.0135097206, 0.285767525, -0.530082881, 0.113298722, -0.129724547, 0.0670884028, 0.149493188, -0.0617235564, -0.238479346, -0.283630252, -0.0588822775, 0.565312803, -0.171043172, -0.10652326, 0.0976450071, 0.534781456, -0.156845704, -0.0480253994, 0.00597760174, 0.449397057, 0.0771201253, 0.344652206, -0.0871425569, 0.345330387, 0.177900821, 0.0390318632, -0.225337446, 0.300412863, 0.286295027, 0.035174489, -0.0743884146, 0.331121832, 0.289069563, -0.168520123, 0.0474938452, 0.156701893, -0.258000255, -0.114123806, -0.0928100646, 0.0624989569, 0.35030064, 0.0171428025, 0.00150060654, -0.287588775, 0.127226189, 0.309583515, -0.030652225, -0.0694010258, 0.178828195, -0.236559704, 0.113749661, -0.12379761, -0.0391594768, 0.317085117, -0.247599423, -0.0250636116, 0.216536433, 0.00525053171, 0.261094034, 0.373894542, 0.256208658, -0.301155508, -0.258028239, -0.0243441351, -0.141106635, 0.523138404, 0.0485578328, -0.0565921366, 0.0685373843, 0.53154707, -0.153182134, 0.0121881068, 0.214072853, -0.0475144126, 0.44517538, 0.0120503651, 0.248578042, 0.444780618, -0.176307604, 0.0653260499, -0.0533154309, 0.0410766266, 0.561017632, 0.379431337, 0.382149428, -0.199403673, -0.0274827089, -0.365465969, 0.332549065, 0.595709443, -0.0261393227, -0.0194830354, 0.573919892, 0.00395603338, -0.214074373, -0.184095159, -0.279999137, -0.299215823, 0.0417990275, 0.295691341, -0.132780015, 0.646226525, -0.349222541, -0.012017875, 0.18422994, 0.0614700988, -0.0295813866, 0.458430082, -0.456961602, -0.154503018, -0.0988531113, 0.625263393, -0.314657658, 0.00507152034, 0.0563785844, 0.590412676, 0.11533422, -0.00469536986, -0.113809466, -0.341424286, -0.281193852, -0.327916861, -0.134057581, -0.238559768, -0.127514705, 0.0890027508, -0.236177027, 0.435842007, -0.130935416, -0.140390649, 0.352221727, -0.121010713, 0.298475653, -0.0214293431, -0.211993009, -0.297033459, -0.186831579, 0.620103717, 0.115540206, -0.177024096, 0.298937589, -0.260433882, -0.186319157, -0.0991054475, -0.170363709, -0.20179674, -0.0838826001, -0.0133801103, 0.30582419, -0.00246372819, -0.133188084, 0.178513736, -0.154469803, 0.252813548, -0.292857885, -0.339029849, 0.0647572875, -0.322565764, 0.189263612, -0.294819474, 0.211947054, 0.251263469, 0.255613655, 0.0804869831, -0.495157987, 0.660171151, 0.234752864, -0.343211293, -0.139396653, 0.0448856018, 0.628873289, -0.206097916, -0.151857197, 0.0876323432, 0.305656523, 0.643062055, -0.179571867, 0.0254980922, 0.467615992, -0.458321154, 0.388876647, 0.205972403, 0.21168837, -0.314859569, -0.295257121, 0.524407327, -0.0496297777, -0.392592728];
    bias_3 : ARRAY[0..23] OF REAL := [0.175584972, -0.123127855, 0, 0, -0.00620653573, -0.0228715166, -0.141794026, -0.0200588796, 0, 0.190223902, 0, -0.0292982291, 0, -0.0160657149, -0.0975855067, 0.225697339, -0.0660655349, -0.0104503827, -0.0145113515, 0.171676457, 0, 0.170017034, -0.00701677147, 0.218090862];

    weights_4 : ARRAY[0..575] OF REAL := [0.536786973, -0.571476996, -0.41954565, -0.30615896, 0.0292444527, -0.00793674123, -0.187810659, -0.306157231, 0.278955013, -0.575931728, 0.19489184, 0.324629754, -0.241611525, -1.03575206, -0.964987397, 0.0663082898, -0.234412253, -0.0820855498, 0.300487906, -0.0394102819, 0.44617027, 0.261538416, -0.367998451, -0.468021899, -0.446363509, -0.164351612, 0.458562702, -0.0304386094, 0.0884533674, 0.613522649, -0.191393808, -0.00453844666, -0.234240249, 0.356710911, -0.534440815, -0.185568437, 0.293668598, 0.429092646, 0.0483992212, -0.469924271, 0.0420621336, 0.300252527, -0.184417844, -0.138343528, -0.0902102664, -0.181992993, 0.446867406, 0.232363895, 0.0150693655, -0.243103772, -0.185197204, 0.194547981, -0.215058848, 0.205206245, -0.00925958157, -0.157177642, -0.246485293, -0.201589465, -0.284912765, 0.0567258596, -0.331246823, 0.105488509, 0.105020255, -0.0127197504, -0.160476819, 0.0676600337, -0.0431795418, -0.224543229, 0.0210678577, 0.172398299, -0.104157582, 0.274997205, 0.122451007, -0.326706767, -0.351181269, 0.122069508, -0.022873193, -0.0581207573, -0.178139463, 0.0562029779, -0.261628568, 0.0177225769, 0.138747662, -0.193212196, -0.0453386307, -0.262532294, -0.240997955, -0.0402922034, 0.148889631, 0.236775368, 0.192761451, -0.0553752184, -0.321817636, -0.0628141463, 0.0567405224, 0.302531928, 0.137698889, 0.0794247687, -0.10497158, 0.230700806, -0.284240723, -0.162641257, 0.0971137583, 0.11107868, 0.304284006, 0.312855959, 0.0705919191, -0.201299161, 0.255538017, -0.0949205756, 0.044130981, -0.0181608312, -0.102627158, -0.295879304, 0.2124587, -0.0965559781, -0.0362335332, 0.168730125, 0.29921332, 0.205723375, 0.0355818942, 0.224375993, 0.294832617, 0.160531193, 0.152477056, 0.324049056, -0.164996684, 0.0887358189, 0.273470521, 0.0712452978, 0.146577194, 0.323198527, 0.346763641, -0.314547539, -0.292661607, 0.00591632165, -0.341849446, -0.283119917, 0.275354981, 0.320525527, 0.0963033214, -0.202617019, 0.182186127, 0.0690234005, -0.679131269, -0.0492588878, 0.164101645, 0.307421893, 0.437007993, 0.537774146, -0.334378421, 0.118354589, -0.207899109, 0.599443316, -0.492537379, 0.0163812041, -0.124113873, -0.0459213965, 0.49334988, -0.165663883, -0.312327683, -0.0646260381, 0.253586382, -0.186140537, -0.484630197, -0.102963001, 0.100501694, 0.342100471, -0.0730798692, 0.0273638275, -0.046032548, -0.279043674, 0.202158853, -0.177257076, -0.188554719, 0.109146774, 0.346752375, 0.294415563, -0.227040142, 0.232832998, 0.269496828, -0.202185765, -0.306152016, -0.208050638, 0.0400530696, 0.23522833, 0.0578660071, 0.243247077, 0.0220626127, -0.279370129, -0.18598558, 0.0541472435, 0.050932616, -0.157867342, -0.275069535, -0.27992031, 0.336847275, -0.305646747, 0.313597769, 0.101961076, 0.113815039, 0.302499563, -0.327620685, -0.195664555, 0.22792998, 0.262621552, 0.180010647, -0.161024302, -0.194168165, 0.329300731, 0.0538795888, -0.252238601, -0.168746457, 0.0946801007, -0.289456725, 0.00608155131, 0.35911876, 0.0764566511, 0.566336691, 0.0153125897, 0.107374318, 0.133425862, 0.200286388, 0.0867452025, 0.381613612, 0.24108766, 0.46200645, -0.259214759, 0.0072132647, -0.099736996, -0.0611620471, -0.179100484, -0.202183485, -0.192014962, -0.00827212259, 0.140485823, 0.285787493, -0.25742659, 0.293467909, 0.307195991, -0.228040576, 0.135603338, 0.237738639, -0.224808589, 0.0356914699, -0.0644816458, -0.215602964, -0.147777557, 0.144645452, 0.247658402, 0.284550756, 0.190389007, -0.0230146945, -0.07220456, 0.229826182, -0.158960462, -0.271376133, -0.204087928, -0.190530732, 0.00172051787, -0.143615812, -0.166735709, 0.0696841776, -0.212757707, -0.72502923, 0.364306897, 0.666826665, 0.0598814376, -0.0481321327, 0.07229577, -0.286086828, 0.13525793, 0.310015291, 0.607683182, -0.260239601, -0.188741758, 0.166386753, 0.214346841, 0.344181389, -0.653774738, -0.104646236, -0.240793377, -0.208343834, 0.102552906, -0.0772212669, -0.324167073, 0.494184285, 0.547423363, -0.272249162, 0.186145872, -0.253451586, -0.1006459, 0.034470886, 0.0575170517, 0.282823056, 0.0104771256, -0.220375329, 0.231437474, -0.0629941225, -0.0971537828, -0.159530371, 0.211183637, 0.0256092548, 0.291559428, -0.28134042, 0.20893988, -0.217550054, -0.00827175379, -0.0406514704, 0.141545624, 0.0761702359, 0.112959802, -0.351895094, -0.0302171111, 0.176429242, 0.311109632, 0.299873829, 0.270576328, 0.007889539, -0.125682995, -0.184819311, 0.286102891, -0.0678215101, -0.192078441, -0.104958385, 0.235353798, 0.219600171, 0.103353798, 0.152216464, -0.278770983, -0.148364156, -0.00862940587, 0.00610713009, -0.220395178, -0.038950514, 0.0999374986, -0.381039023, 0.215833709, 0.635107338, -0.391911983, 0.31318441, -0.0982320681, 0.155621529, -0.0327736437, 0.375541598, 0.604466379, -0.256146878, -0.203460529, -0.0318981707, 0.060248062, 0.361447066, -0.252633393, 0.320484608, -0.10533829, -0.304791301, -0.292700469, 0.021918444, -0.0490716472, 0.51709801, 0.169388801, -0.050713256, -0.137047842, -0.356132329, -0.267450601, 0.221725002, -0.0675771758, -0.0170709342, -0.0522325039, 0.622837245, 0.199781016, 0.479887038, 0.179646462, 0.249492973, -0.449901342, -0.631632686, 0.148131013, -0.145344928, 0.274162978, -0.0622148886, 0.0685222074, 0.0551666059, 0.354044527, -0.0923385769, 0.0325434208, -0.68811202, 0.0934957266, 0.655678689, 0.265559822, -0.229217127, 0.542057216, 0.0905142426, -0.207350105, -0.393493563, 0.660121799, -0.491635948, -0.0963397622, -0.00393542647, 0.379227102, 0.120349266, -0.638450325, -0.193138272, 0.100851685, -0.104843296, -0.287845194, -0.600140333, 0.0626947805, 0.564362764, 0.574099183, -0.107015058, -0.189990997, -0.130377576, -0.348115563, 0.316623598, 0.362836152, 0.193917304, -0.339228332, -0.187139511, 0.161454126, 0.158694118, -0.0982089937, -0.00619760156, 0.287415713, -0.179751784, 0.155939788, -0.0470742285, 0.157508224, -0.0908677578, 0.0169253349, 0.0398236364, 0.223295718, -0.149136379, 0.337734401, 0.0509377234, -0.121674545, -0.0781851709, -0.116671577, 0.150503129, 0.0782350525, -0.009878546, -0.344213039, 0.295079112, 0.186227053, -0.0153816687, -0.165958524, -0.207513541, -0.107627325, 0.297569245, -0.107240297, -0.294790298, -0.12299116, -0.13974835, -0.349520981, 0.334641427, -0.315597594, -0.351451486, -0.0497232378, 0.523416281, -0.150883317, -0.430363595, 0.283077687, 0.368172526, -0.426088572, 0.225863934, -0.281553745, 0.409919202, -0.491759449, 0.557659686, -0.207404137, -0.0486885309, -0.59106946, -0.669140458, 0.397414953, -0.0522342026, -0.211202741, -0.285691649, 0.12049748, 0.677952349, 0.664889336, -0.0535091497, -0.385653973, -0.0901891887, -0.171689659, 0.154431134, 0.0888457298, -0.0334436893, -0.00624498725, -0.290563494, -0.256944895, -0.131268963, -0.221912593, 0.166501731, -0.120807528, -0.313281566, 0.204365104, -0.0267566741, -0.208927408, -0.241888523, 0.121474385, 0.291662663, 0.343239278, 0.157343894, 0.0052857995, 0.0702802837, 0.228197545, -0.1296601, -0.11545413, 0.544608831, -0.105114311, 0.246841788, 0.460096389, -0.3347058, -0.147451848, 0.0235350896, 0.325939119, 0.302343696, -0.185763747, -0.195407376, 0.206940651, 0.0175213888, -0.00879597198, -0.0931996703, -0.222991973, 0.0488129258, -0.299850702, 0.205607086, 0.315567046, 0.375953585, 0.493875355, 0.200358972, -0.142462894, -0.290279835, 0.145780712, -0.289276242, -0.185444608, -0.120101064, -0.0401476622, -0.0894734785, -0.00486295065, -0.322057813, -0.239333481, -0.160521746, 0.263630539, 0.236000866, 0.0357191265, -0.0323565602, 0.17025134, 0.136110738, -0.340670377, 0.126549229, 0.0283196718, 0.178190753, -0.0187530816, 0.253103286, -0.0749137104, -0.343879074, -0.147712111, 0.508385301, -0.346718282, -0.0123189902, -0.340981901, 0.475469053, 0.135450944, 0.625618577, -0.0120549202, -0.0878968239, -0.254162699, -0.115267202, 0.260036558, -0.177432582, -0.295926511, 0.154717222, 0.0635785088, 0.613382041, 0.736293197, -0.0829628482, -0.224064127];
    bias_4 : ARRAY[0..23] OF REAL := [0.0884786695, -0.113101497, 0.0612285659, -0.0210166965, 0.120523497, -0.0150198843, -0.0184283908, 0, 0.219995826, -0.0337756053, 0.168627232, 0, 0, -0.153112203, -0.154962838, 0.0574183092, 0, 0, -0.00937702879, -0.0990674496, 0.219536304, 0.193301007, -0.100828946, 0.0894805416];

    weights_5 : ARRAY[0..71] OF REAL := [0.790903628, -0.415320307, -0.231604829, 0.27451545, 0.0347574018, 0.557182014, -0.888507545, 0.0090645412, 0.146589607, -0.325830609, 0.44091019, -0.170073912, -0.181570187, 0.356534123, -0.338704884, -0.588768303, 0.111096844, 0.603150606, -0.213561445, 0.298852831, 0.0858602077, -0.020580709, 0.140703827, 0.174954027, 0.111611515, 0.333741456, -0.732370794, -0.721106887, 0.373889863, 0.34062323, 0.676797688, -0.0135949906, -1.02032185, -0.300230086, -0.0818669498, 0.239884347, 0.372507244, 0.162670761, -0.0934614837, -0.37575525, -0.75501436, 0.594942093, -0.194047213, -0.701864243, 0.769190073, 0.759077191, -0.926579118, 0.248977929, -0.1242823, 0.3033382, -0.441861033, 0.351782233, 0.202550083, -0.390180916, 0.226951405, 0.236660749, 0.227680445, 0.102284789, 0.265807033, 0.147111937, 0.0562378019, -0.202766195, -0.96057111, 0.327031195, 0.207056925, -0.815793455, -0.0683416873, 0.367274374, 0.337488323, -0.801836371, 0.0764635578, 0.168529764];
    bias_5 : ARRAY[0..2] OF REAL := [0.0512467474, 0.106338561, -0.171999738];

END_VAR

VAR
    (* Merged variables from all regions *)
    buffer_0 : ARRAY[0..23] OF REAL;
    buffer_1 : ARRAY[0..23] OF REAL;

    (* Temporary computation variables *)
    i : DINT;
    j : DINT;
    t : DINT;
    sum : REAL;
    (* Computation helpers *)
    max_val : REAL;
    exp_val : REAL;
    exp_sum : REAL;
    (* Spatial loop variables *)
    oc : DINT;
    oh : DINT;
    ow : DINT;
    ic : DINT;
    kh : DINT;
    kw : DINT;
    ih : DINT;
    iw : DINT;
END_VAR

(* Forward pass execution *)

(* Region: r0 [ACYCLIC] *)
(* Acyclic Region r0 *)
(* Layer 0: Fused Linear + RELU *)
FOR j := 0 TO 23 DO
    sum := 0.0;
    FOR i := 0 TO 0 DO
        sum := sum + input_data * weights_0[i * 24 + j];
    END_FOR;
buffer_1[j] := MAX(sum + bias_0[j], 0.0);
END_FOR;

(* Layer 1: Fused Linear + RELU *)
FOR j := 0 TO 23 DO
    sum := 0.0;
    FOR i := 0 TO 23 DO
        sum := sum + buffer_1[i] * weights_1[i * 24 + j];
    END_FOR;
buffer_0[j] := MAX(sum + bias_1[j], 0.0);
END_FOR;

(* Layer 2: Fused Linear + RELU *)
FOR j := 0 TO 23 DO
    sum := 0.0;
    FOR i := 0 TO 23 DO
        sum := sum + buffer_0[i] * weights_2[i * 24 + j];
    END_FOR;
buffer_1[j] := MAX(sum + bias_2[j], 0.0);
END_FOR;

(* Layer 3: Fused Linear + RELU *)
FOR j := 0 TO 23 DO
    sum := 0.0;
    FOR i := 0 TO 23 DO
        sum := sum + buffer_1[i] * weights_3[i * 24 + j];
    END_FOR;
buffer_0[j] := MAX(sum + bias_3[j], 0.0);
END_FOR;

(* Layer 4: Fused Linear + RELU *)
FOR j := 0 TO 23 DO
    sum := 0.0;
    FOR i := 0 TO 23 DO
        sum := sum + buffer_0[i] * weights_4[i * 24 + j];
    END_FOR;
buffer_1[j] := MAX(sum + bias_4[j], 0.0);
END_FOR;

(* Layer 5: Fused Linear + SOFTMAX *)
FOR j := 0 TO 2 DO
    sum := 0.0;
    FOR i := 0 TO 23 DO
        sum := sum + buffer_1[i] * weights_5[i * 3 + j];
    END_FOR;
output_data[j] := sum + bias_5[j];
END_FOR;

(* Softmax: find max *)
max_val := output_data[0];
FOR i := 1 TO 2 DO
    IF output_data[i] > max_val THEN
        max_val := output_data[i];
    END_IF;
END_FOR;

(* Softmax: compute exponentials and sum *)
exp_sum := 0.0;
FOR i := 0 TO 2 DO
    output_data[i] := EXP(output_data[i] - max_val);
    exp_sum := exp_sum + output_data[i];
END_FOR;

(* Softmax: normalize *)
FOR i := 0 TO 2 DO
    output_data[i] := output_data[i] / exp_sum;
END_FOR;

END_FUNCTION_BLOCK
